// TIA Portal project "Project2" (V19)

(* hardware
DEVICE "ET 200SP station_1"  ET 200SP-Station
   slot 0: "IO device_1"  IM 155-6 PN ST  6ES7 155-6AU01-0BN0  V4.2
   slot 0: "Rack_0"  Rack  6ES5 710-8MAx1
   slot 1: "AI 4xRTD/TC 2-/3-/4-wire HF_1"  AI 4xRTD/TC 2-,3-,4-wire HF  6ES7 134-6JD00-0CA1  V2.1
      slot 1: "AI 4xRTD/TC 2-/3-/4-wire HF_1"  AI 4xRTD/TC 2-,3-,4-wire HF
   slot 2: "TM Count 1x24V_1"  TM Count 1x24V  6ES7 138-6AA01-0BA0  V2.0
      slot 1: "TM Count 1x24V_1"  TM Count 1x24V
   slot 127: "BA 2xRJ45"  BA 2xRJ45  6ES7 193-6AR00-0AA0  V0.0
      slot 1: "Port_1"  X1 P1 R  6ES7 193-6AR00-0AA0  V0.0
      slot 2: "Port_2"  X1 P2 R  6ES7 193-6AR00-0AA0  V0.0
DEVICE "ET 200SP station_2"  ET 200SP-Station
   slot 0: "Rack_0"  Rack  6ES5 710-8MAx1
   slot 1: "PLC_1"  CPU 1512SP-1 PN  6ES7 512-1DM03-0AB0  V3.1
      slot 32768: "PROFINET interface_1"  X1
         slot 32771: "Port_3"  X1 P3
   slot 2: "TM Count 1x24V_1"  TM Count 1x24V  6ES7 138-6AA01-0BA0  V2.0
      slot 1: "TM Count 1x24V_1"  TM Count 1x24V
   slot 127: "BA 2xRJ45"  BA 2xRJ45  6ES7 193-6AR00-0AA0  V0.0
      slot 32769: "Port_1"  X1 P1  6ES7 193-6AR00-0AA0
      slot 32770: "Port_2"  X1 P2  6ES7 193-6AR00-0AA0
*)

// ===== PLC "PLC_1"  CPU 1512SP-1 PN =====

ORGANIZATION_BLOCK "Main"   // OB1, LAD, ProgramCycle
TITLE = "Main Program Sweep (Cycle)"
{ S7_Optimized_Access := 'TRUE' }
VERSION : 0.1
   VAR_INPUT
      Initial_Call : Bool;   // Initial call of this OB
      Remanence : Bool;   // =True, if remanent data are available
   END_VAR
BEGIN
END_ORGANIZATION_BLOCK